// LS Electric XG5000 project: 8_29
// PLC LSPLC
// module base 0 slot 0: 입출력 모듈:XBC-DR14E (DC 24V 입력 8점, 릴레이 출력 6점)

PROGRAM NewProgram (task: 스캔 프로그램)

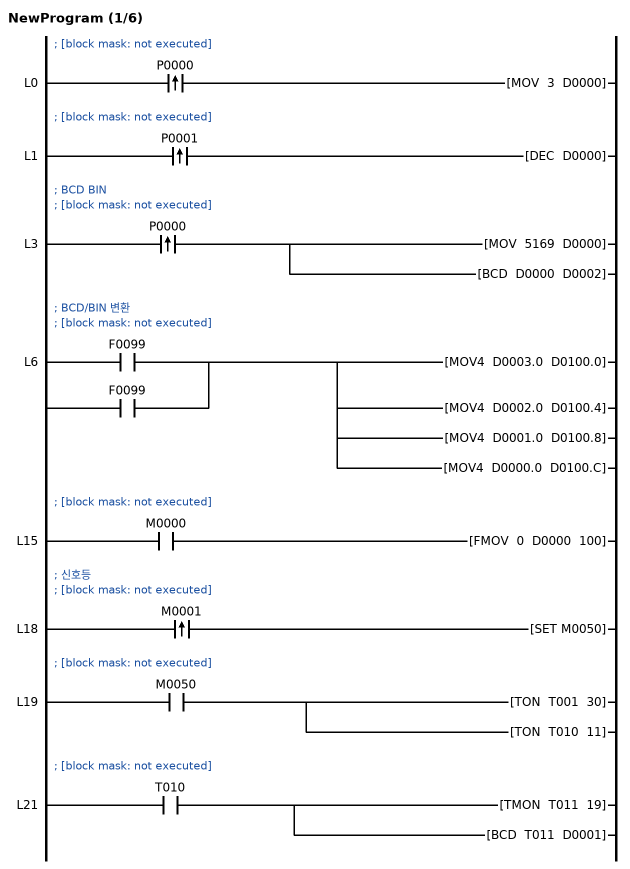
; L0 (block mask: not executed)
LOADP     P0000
MOV       3 D0000
; L1 (block mask: not executed)
LOADP     P0001
DEC       D0000
// BCD BIN
; L3 (block mask: not executed)
LOADP     P0000
MOV       5169 D0000
BCD       D0000 D0002
// BCD/BIN 변환
; L6 (block mask: not executed)
LOAD      F0099
OR        F0099
MOV4      D0003.0 D0100.0
MOV4      D0002.0 D0100.4
MOV4      D0001.0 D0100.8
MOV4      D0000.0 D0100.C
; L15 (block mask: not executed)
LOAD      M0000
FMOV      0 D0000 100
// 신호등
; L18 (block mask: not executed)
LOADP     M0001
SET       M0050
; L19 (block mask: not executed)
LOAD      M0050
TON       T001 30
TON       T010 11
; L21 (block mask: not executed)
LOAD      T010
TMON      T011 19
BCD       T011 D0001

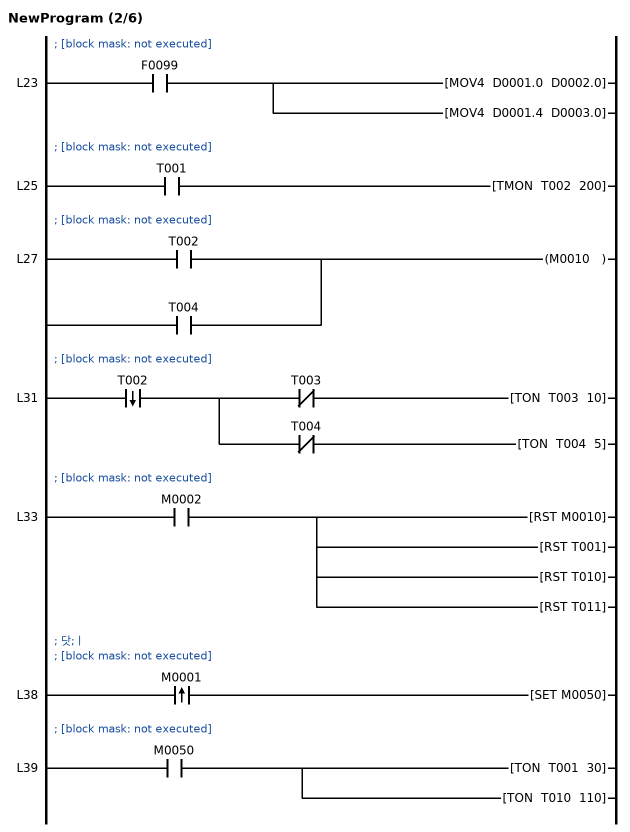
; L23 (block mask: not executed)
LOAD      F0099
MOV4      D0001.0 D0002.0
MOV4      D0001.4 D0003.0
; L25 (block mask: not executed)
LOAD      T001
TMON      T002 200
; L27 (block mask: not executed)
LOAD      T002
OR        T004
OUT       M0010
; L31 (block mask: not executed)
LOADN     T002
MPUSH
AND NOT   T003
TON       T003 10
MPOP
AND NOT   T004
TON       T004 5
; L33 (block mask: not executed)
LOAD      M0002
RST       M0010
RST       T001
RST       T010
RST       T011
// 닷;ㅣ
; L38 (block mask: not executed)
LOADP     M0001
SET       M0050
; L39 (block mask: not executed)
LOAD      M0050
TON       T001 30
TON       T010 110

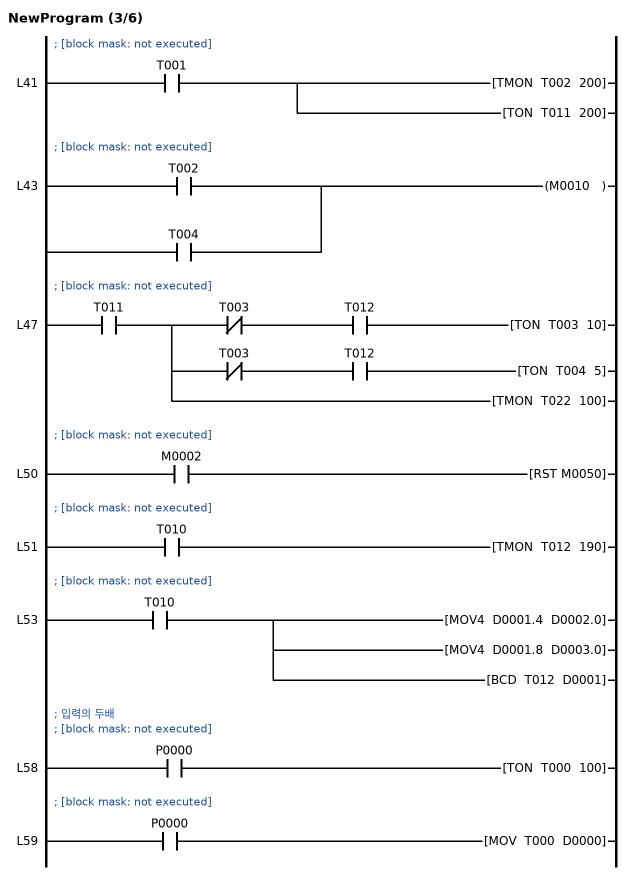
; L41 (block mask: not executed)
LOAD      T001
TMON      T002 200
TON       T011 200
; L43 (block mask: not executed)
LOAD      T002
OR        T004
OUT       M0010
; L47 (block mask: not executed)
LOAD      T011
MPUSH
AND NOT   T003
AND       T012
TON       T003 10
MLOAD
AND NOT   T003
AND       T012
TON       T004 5
MPOP
TMON      T022 100
; L50 (block mask: not executed)
LOAD      M0002
RST       M0050
; L51 (block mask: not executed)
LOAD      T010
TMON      T012 190
; L53 (block mask: not executed)
LOAD      T010
MOV4      D0001.4 D0002.0
MOV4      D0001.8 D0003.0
BCD       T012 D0001
// 입력의 두배
; L58 (block mask: not executed)
LOAD      P0000
TON       T000 100
; L59 (block mask: not executed)
LOAD      P0000
MOV       T000 D0000

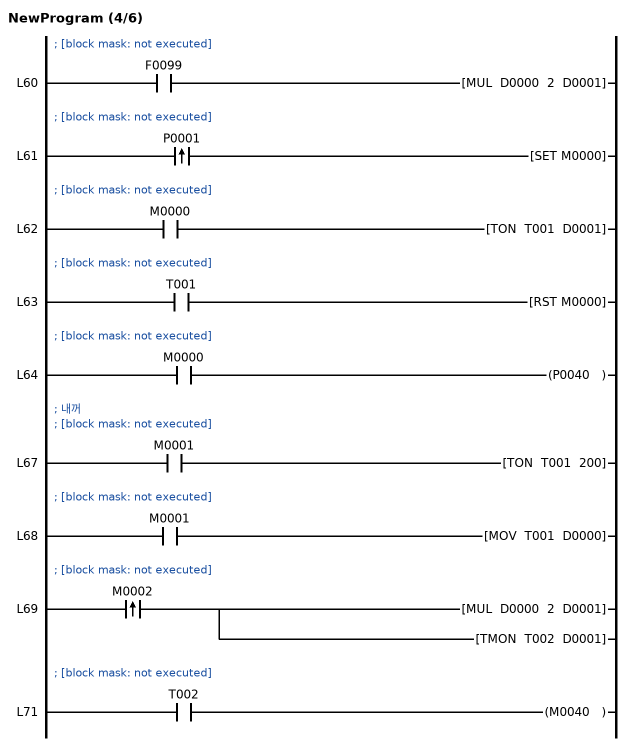
; L60 (block mask: not executed)
LOAD      F0099
MUL       D0000 2 D0001
; L61 (block mask: not executed)
LOADP     P0001
SET       M0000
; L62 (block mask: not executed)
LOAD      M0000
TON       T001 D0001
; L63 (block mask: not executed)
LOAD      T001
RST       M0000
; L64 (block mask: not executed)
LOAD      M0000
OUT       P0040
// 내꺼
; L67 (block mask: not executed)
LOAD      M0001
TON       T001 200
; L68 (block mask: not executed)
LOAD      M0001
MOV       T001 D0000
; L69 (block mask: not executed)
LOADP     M0002
MUL       D0000 2 D0001
TMON      T002 D0001
; L71 (block mask: not executed)
LOAD      T002
OUT       M0040

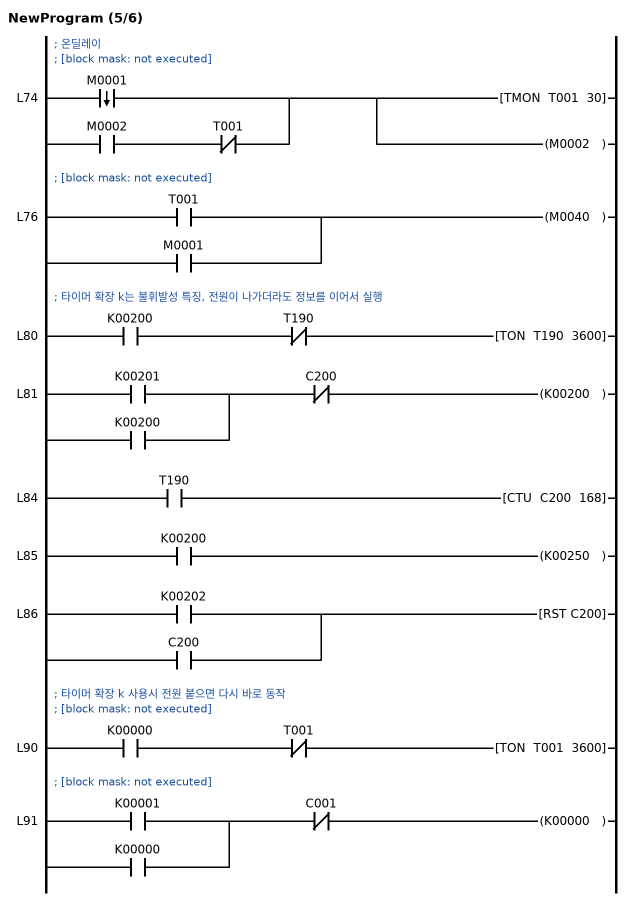
// 온딜레이
; L74 (block mask: not executed)
LOADN     M0001
LOAD      M0002
AND NOT   T001
OR LOAD
TMON      T001 30
OUT       M0002
; L76 (block mask: not executed)
LOAD      T001
OR        M0001
OUT       M0040
// 타이머 확장 k는 불휘발성 특징, 전원이 나가더라도 정보를 이어서 실행
; L80
LOAD      K00200
AND NOT   T190
TON       T190 3600
; L81
LOAD      K00201
OR        K00200
AND NOT   C200
OUT       K00200
; L84
LOAD      T190
CTU       C200 168
; L85
LOAD      K00200
OUT       K00250
; L86
LOAD      K00202
OR        C200
RST       C200
// 타이머 확장 k 사용시 전원 붙으면 다시 바로 동작
; L90 (block mask: not executed)
LOAD      K00000
AND NOT   T001
TON       T001 3600
; L91 (block mask: not executed)
LOAD      K00001
OR        K00000
AND NOT   C001
OUT       K00000

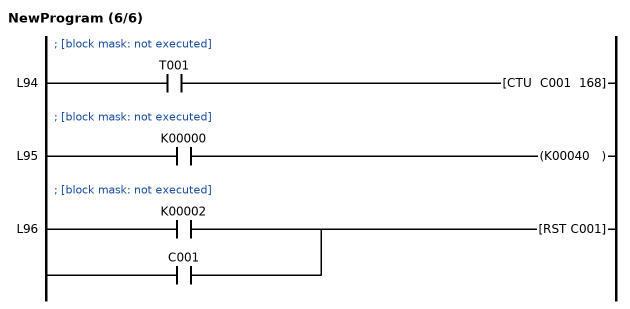
; L94 (block mask: not executed)
LOAD      T001
CTU       C001 168
; L95 (block mask: not executed)
LOAD      K00000
OUT       K00040
; L96 (block mask: not executed)
LOAD      K00002
OR        C001
RST       C001